FUNCTION_BLOCK Error_Merge (* Basic FB with empty ECC *)
  (* Standard: 61499-2 *)
  (* Version 1.0, 2023-03-17, AK125171 *)
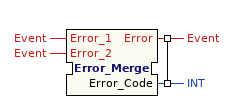
  EVENT_INPUT
    Error_1;
    Error_2;
  END_EVENT
  EVENT_OUTPUT
    Error WITH Error_Code;
  END_EVENT
  VAR_OUTPUT
    Error_Code : INT;
  END_VAR
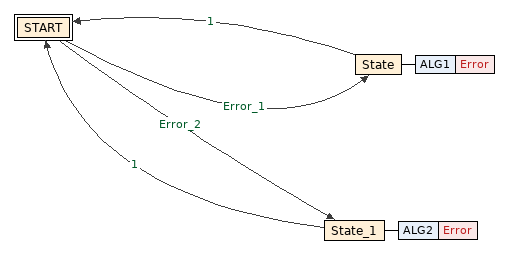
  EC_STATES
    START; (* Initial State *)
    State : ALG1 -> Error;
    State_1 : ALG2 -> Error;
  END_STATES
  EC_TRANSITIONS
    START TO State := Error_1;
    START TO State_1 := Error_2;
    State TO START := 1;
    State_1 TO START := 1;
  END_TRANSITIONS
  ALGORITHM ALG1 IN ST:
Error_Code:=1;
  END_ALGORITHM
  ALGORITHM ALG2 IN ST:
Error_Code:=2;
  END_ALGORITHM
END_FUNCTION_BLOCK
